TYPE SampleTaskFunctionBuffer : STRUCT
    x : LREAL;
    y : LREAL;
END_STRUCT
END_TYPE

(* stored: Version 1.1.0.1, ProductVersion 3.1.4024.6
   DUT SampleTaskFunctionBuffer: Id {056d4909-fab7-493d-b7d6-9ed7ad026b81} *)
